// Mitsubishi GX Works2 project: PLC_GROUP_02   PLC: FX3G
// PLC_GROUP_02

// global labels: Global1
VAR_GLOBAL
  sw5 AT X005 : BOOL;
  light7 AT Y007 : BOOL;
  ts1 AT TS1 : BOOL;
  light1 AT Y001 : BOOL;
  ts2 AT TS2 : BOOL;
  inventoryRaspberry AT D1102 : INT;
  inventoryLemon AT D1104 : INT;
  inventoryStabilizer AT D1106 : INT;
  inventoryGummy AT D1108 : INT;
  sw3 AT X003 : BOOL;
  light2 AT Y002 : BOOL;
  anlogInput1 AT D8280 : INT;
  helper11 AT M11 : ARRAY [0..2] OF BOOL;
  regularGummy AT M12 : BOOL;
  luxeryGummy AT M13 : BOOL;
  tc1 AT TC1 : BOOL;
  tempDetected AT M5 : BOOL;
  tc2 AT TC2 : BOOL;
END_VAR
VAR_GLOBAL CONSTANT
  constant0 : INT;
  constant5 : INT := 5;
END_VAR
VAR_GLOBAL
  light0 AT Y000 : BOOL;
END_VAR
VAR_GLOBAL CONSTANT
  needRaspberryReg : INT := 280;
  needLemonReg : INT := 455;
  needStabilizerReg : INT := 105;
  needGummyReg : INT := 28;
  needRaspberryLux : INT := 385;
  needLemonLux : INT := 665;
  needStabilizerLux : INT := 210;
  needGummyLux : INT := 70;
  lemonAndRaspberryMake : INT := 10;
  LemRasMaking : INT := 50;
END_VAR
VAR_GLOBAL
  cooling AT X002 : BOOL;
  temp AT D1130 : INT;
END_VAR
VAR_GLOBAL CONSTANT
  twoCoolingTime : INT := 160;
  onePackage : INT := 1;
  byTen : REAL := 10.0;
END_VAR
VAR_GLOBAL
  inventory AT M1 : BOOL;
  emergency AT X005 : BOOL;
  chooseType AT X001 : BOOL;
  determineType AT M11 : ARRAY [0..2] OF BOOL;
  noInvantoryRegular AT M4 : BOOL;
  noInvantoryLux AT M6 : BOOL;
  tempSensor AT X003 : BOOL;
  startD AT X007 : BOOL;
  helper0 AT M0 : BOOL;
  ts3 AT TS3 : BOOL;
  tc3 AT TC3 : BOOL;
END_VAR
VAR_GLOBAL CONSTANT
  mixingTimeReg : INT := 30;
END_VAR
VAR_GLOBAL
  light5 AT Y005 : BOOL;
  ts4 AT TS4 : BOOL;
  light6 AT Y006 : BOOL;
  tc4 AT TC4 : BOOL;
  tc5 AT TC5 : BOOL;
  tc6 AT TC6 : BOOL;
END_VAR
VAR_GLOBAL CONSTANT
  mixingTimelux : INT := 50;
END_VAR
VAR_GLOBAL
  ts5 AT TS5 : BOOL;
  ts6 AT TS6 : BOOL;
END_VAR
VAR_GLOBAL CONSTANT
  flickeringTime : INT := 5;
END_VAR
VAR_GLOBAL
  last AT M13 : BOOL;
  first AT M1 : BOOL;
  restAllM AT M14 : BOOL;
END_VAR
VAR_GLOBAL CONSTANT
  lessThen5 : INT := 5;
  con0 : INT;
  con5 : INT := 5;
  con6 : INT := 6;
  con10 : INT := 10;
  conFlote10 : REAL := 10.0;
  con40 : INT := 40;
  con400 : INT := 400;
END_VAR
VAR_GLOBAL
  sampleInput AT M2 : BOOL;
  endOfDay AT M3 : BOOL;
  analogOut AT D8282 : INT;
  packages AT D1130 : INT;
  endOfDaytPack AT D1132 : INT;
  analogInputDiv AT D1140 : INT;
  coolingCont AT D1142 : INT;
END_VAR
VAR_GLOBAL CONSTANT
  rasRegGram : INT := 350;
END_VAR
VAR_GLOBAL
  finishFirstCooling AT M7 : BOOL;
END_VAR
VAR_GLOBAL CONSTANT
  limRegGram : INT := 490;
  coolingTime : INT := 80;
END_VAR
VAR_GLOBAL
  mixingCont AT D1144 : INT;
END_VAR
VAR_GLOBAL CONSTANT
  con868 : INT := 868;
  con1330 : INT := 1330;
END_VAR
VAR_GLOBAL
  coolingContRas AT D1142 : INT;
  coolingContlim AT D1146 : INT;
END_VAR
VAR_GLOBAL CONSTANT
  limLuxGram : INT := 700;
  rasLuxGram : INT := 560;
END_VAR
VAR_GLOBAL
  stopDay AT M20 : BOOL;
  firstD AT D1102 : INT;
  lastD AT D1130 : INT;
  first2D AT D1134 : INT;
  last2D AT D1146 : INT;
  startMixing AT M8 : BOOL;
END_VAR

// task Task_01 (event TRUE, interval 0, priority 31): POU_01

PROGRAM POU_01
(* structured ladder/FBD written out as ST: instructions are called as NAME(EN, inputs, outputs); _pN, _eN, _tN stand for wires *)
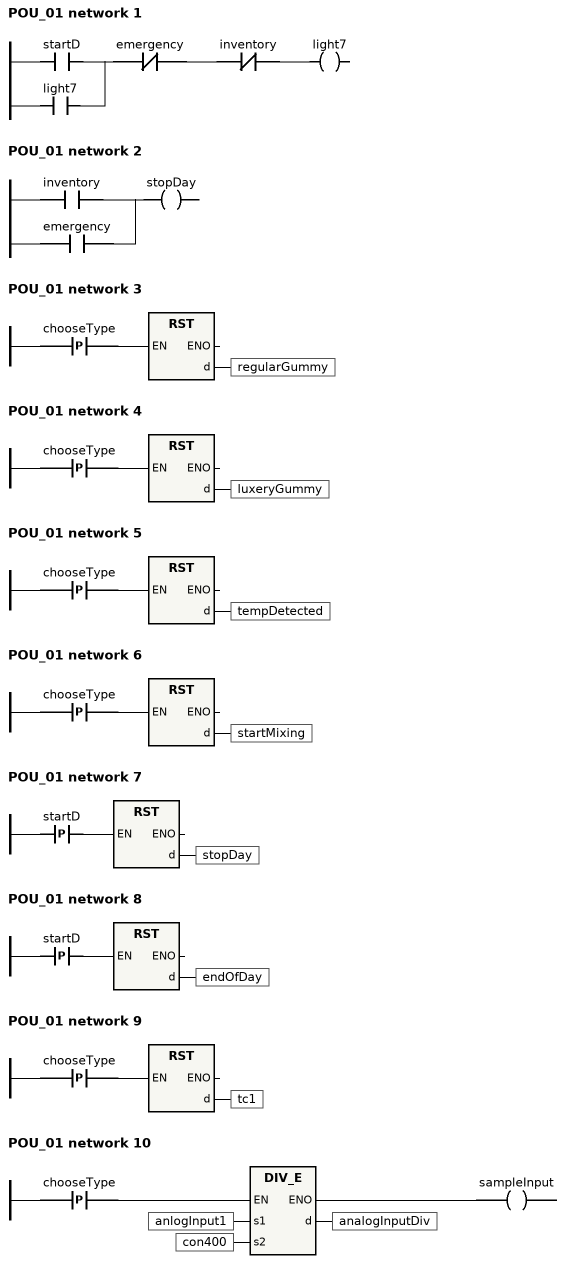
(* network 1 *)
light7 := ((startD OR light7) AND NOT emergency) AND NOT inventory;
(* network 2 *)
stopDay := inventory OR emergency;
(* network 3 *)
RST(LDP(TRUE, chooseType), regularGummy);
(* network 4 *)
RST(LDP(TRUE, chooseType), luxeryGummy);
(* network 5 *)
RST(LDP(TRUE, chooseType), tempDetected);
(* network 6 *)
RST(LDP(TRUE, chooseType), startMixing);
(* network 7 *)
RST(LDP(TRUE, startD), stopDay);
(* network 8 *)
RST(LDP(TRUE, startD), endOfDay);
(* network 9 *)
RST(LDP(TRUE, chooseType), tc1);
(* network 10 *)
_e1 := DIV_E(LDP(TRUE, chooseType), anlogInput1, con400, analogInputDiv);
sampleInput := _e1;
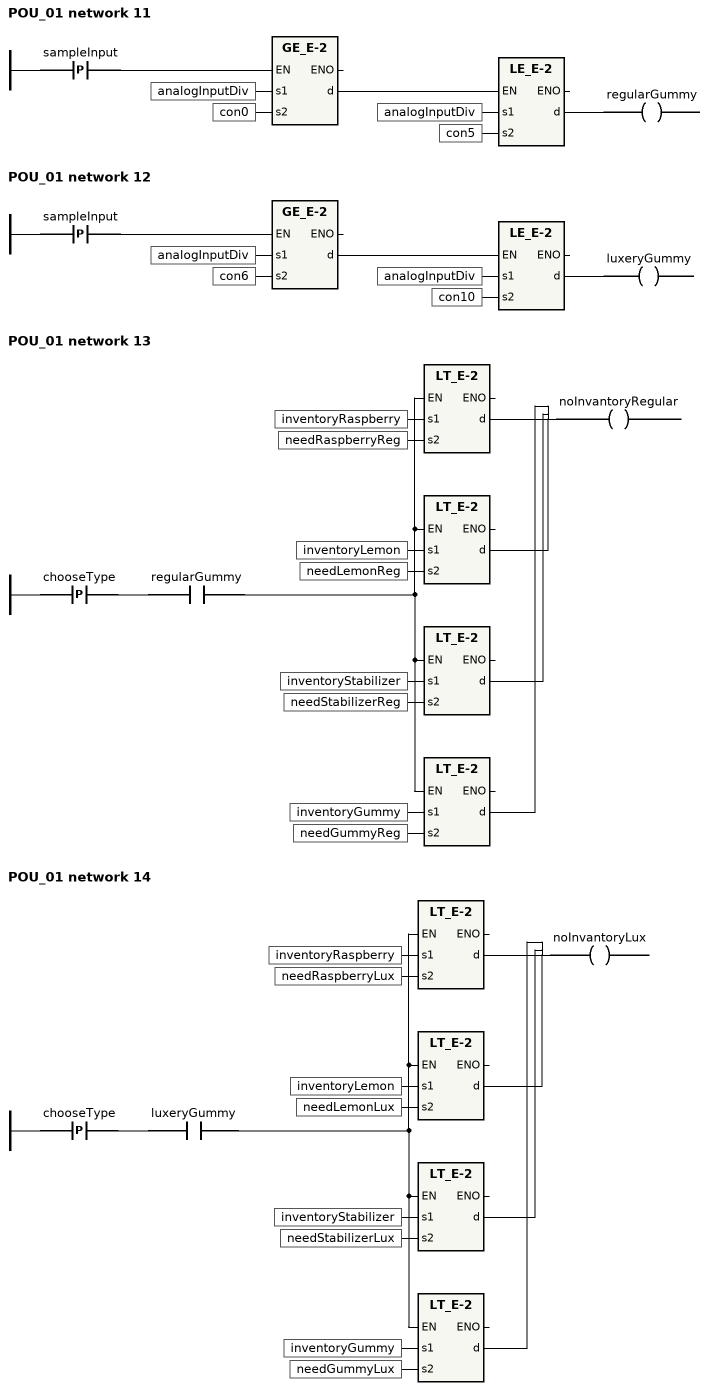
(* network 11 *)
GE_E(LDP(TRUE, sampleInput), analogInputDiv, con0, _t1);
LE_E(_t1, analogInputDiv, con5, _t2);
regularGummy := _t2;
(* network 12 *)
GE_E(LDP(TRUE, sampleInput), analogInputDiv, con6, _t1);
LE_E(_t1, analogInputDiv, con10, _t2);
luxeryGummy := _t2;
(* network 13 *)
_p1 := LDP(TRUE, chooseType) AND regularGummy;
LT_E(_p1, inventoryRaspberry, needRaspberryReg, _t2);
LT_E(_p1, inventoryLemon, needLemonReg, _t3);
LT_E(_p1, inventoryStabilizer, needStabilizerReg, _t4);
LT_E(_p1, inventoryGummy, needGummyReg, _t5);
noInvantoryRegular := _t2 OR _t3 OR _t4 OR _t5;
(* network 14 *)
_p1 := LDP(TRUE, chooseType) AND luxeryGummy;
LT_E(_p1, inventoryRaspberry, needRaspberryLux, _t2);
LT_E(_p1, inventoryLemon, needLemonLux, _t3);
LT_E(_p1, inventoryStabilizer, needStabilizerLux, _t4);
LT_E(_p1, inventoryGummy, needGummyLux, _t5);
noInvantoryLux := _t2 OR _t3 OR _t4 OR _t5;
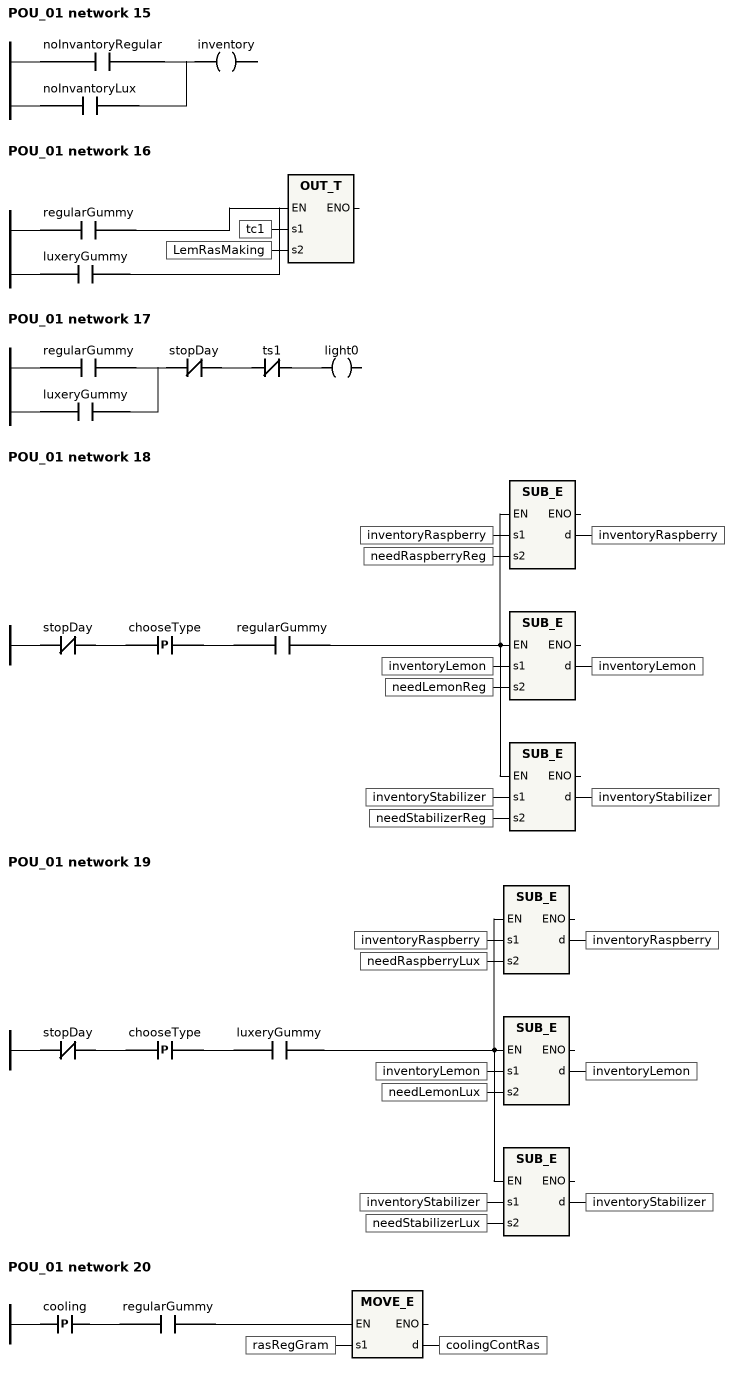
(* network 15 *)
inventory := noInvantoryRegular OR noInvantoryLux;
(* network 16 *)
OUT_T(regularGummy OR luxeryGummy, tc1, LemRasMaking);
(* network 17 *)
light0 := ((regularGummy OR luxeryGummy) AND NOT stopDay) AND NOT ts1;
(* network 18 *)
_p1 := NOT stopDay AND LDP(TRUE, chooseType) AND regularGummy;
SUB_E(_p1, inventoryRaspberry, needRaspberryReg, inventoryRaspberry);
SUB_E(_p1, inventoryLemon, needLemonReg, inventoryLemon);
SUB_E(_p1, inventoryStabilizer, needStabilizerReg, inventoryStabilizer);
(* network 19 *)
_p1 := NOT stopDay AND LDP(TRUE, chooseType) AND luxeryGummy;
SUB_E(_p1, inventoryRaspberry, needRaspberryLux, inventoryRaspberry);
SUB_E(_p1, inventoryLemon, needLemonLux, inventoryLemon);
SUB_E(_p1, inventoryStabilizer, needStabilizerLux, inventoryStabilizer);
(* network 20 *)
MOVE_E(LDP(TRUE, cooling) AND regularGummy, rasRegGram, coolingContRas);
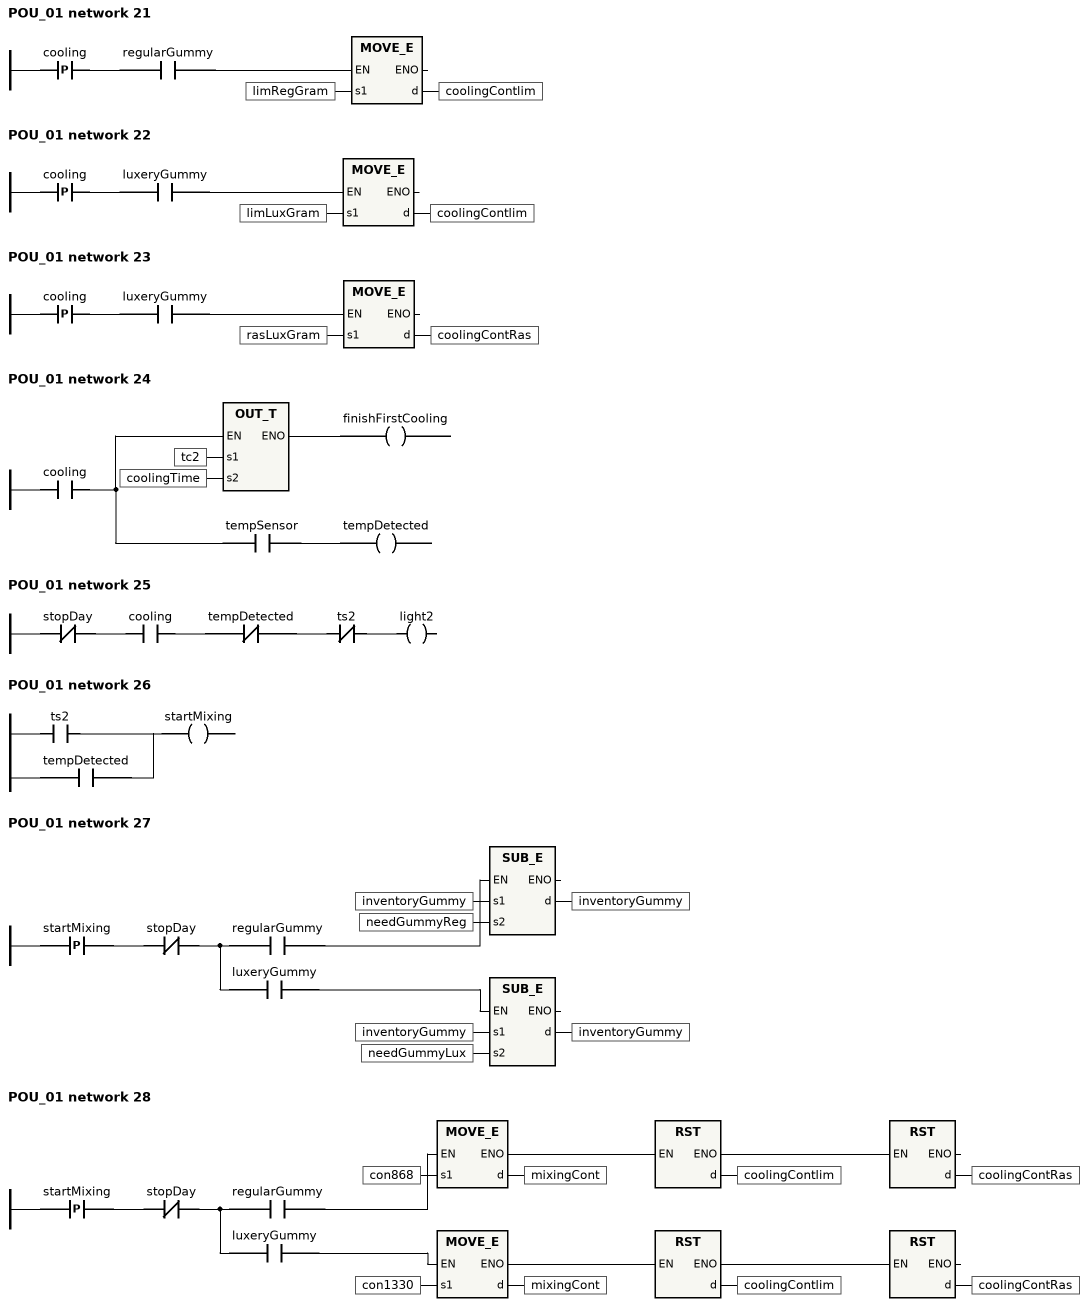
(* network 21 *)
MOVE_E(LDP(TRUE, cooling) AND regularGummy, limRegGram, coolingContlim);
(* network 22 *)
MOVE_E(LDP(TRUE, cooling) AND luxeryGummy, limLuxGram, coolingContlim);
(* network 23 *)
MOVE_E(LDP(TRUE, cooling) AND luxeryGummy, rasLuxGram, coolingContRas);
(* network 24 *)
_e1 := OUT_T(cooling, tc2, coolingTime);
finishFirstCooling := _e1;
tempDetected := cooling AND tempSensor;
(* network 25 *)
light2 := NOT stopDay AND cooling AND NOT tempDetected AND NOT ts2;
(* network 26 *)
startMixing := ts2 OR tempDetected;
(* network 27 *)
_p1 := LDP(TRUE, startMixing) AND NOT stopDay;
SUB_E(_p1 AND regularGummy, inventoryGummy, needGummyReg, inventoryGummy);
SUB_E(_p1 AND luxeryGummy, inventoryGummy, needGummyLux, inventoryGummy);
(* network 28 *)
_p1 := LDP(TRUE, startMixing) AND NOT stopDay;
_e2 := MOVE_E(_p1 AND regularGummy, con868, mixingCont);
_e3 := RST(_e2, coolingContlim);
RST(_e3, coolingContRas);
_e4 := MOVE_E(_p1 AND luxeryGummy, con1330, mixingCont);
_e5 := RST(_e4, coolingContlim);
RST(_e5, coolingContRas);
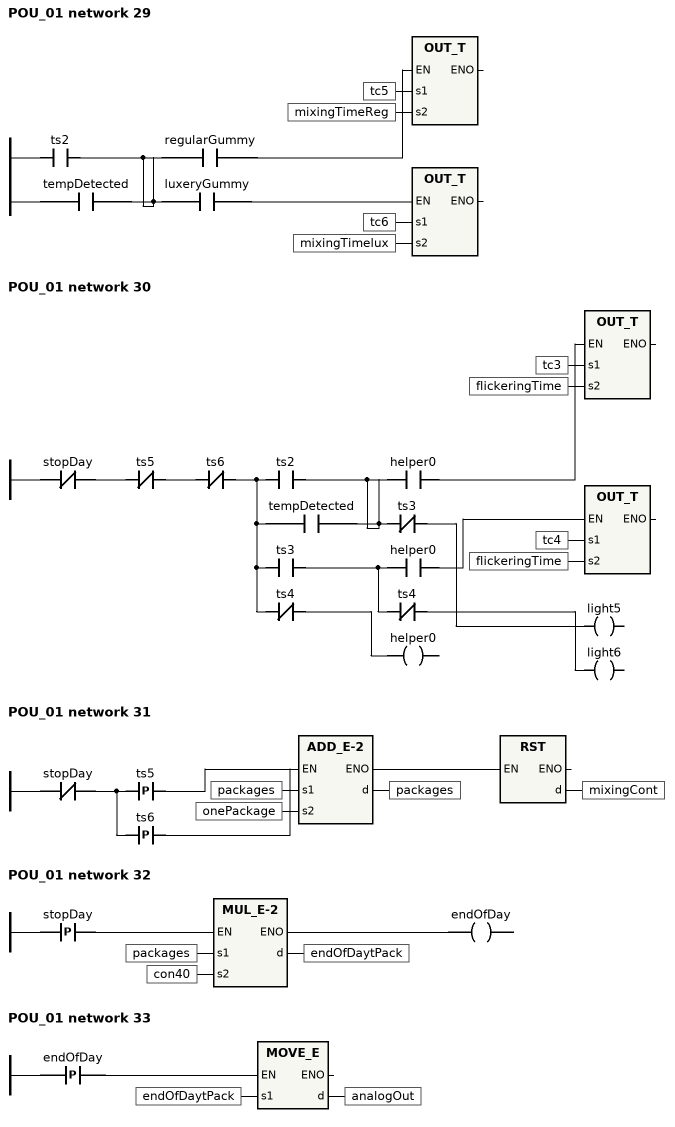
(* network 29 *)
_p1 := ts2 OR tempDetected;
OUT_T(_p1 AND regularGummy, tc5, mixingTimeReg);
OUT_T(_p1 AND luxeryGummy, tc6, mixingTimelux);
(* network 30 *)
_p1 := NOT stopDay AND NOT ts5 AND NOT ts6;
_p2 := (_p1 AND ts2) OR (_p1 AND tempDetected);
OUT_T(_p2 AND helper0, tc3, flickeringTime);
light5 := _p2 AND NOT ts3;
_p3 := _p1 AND ts3;
OUT_T(_p3 AND helper0, tc4, flickeringTime);
light6 := _p3 AND NOT ts4;
helper0 := _p1 AND NOT ts4;
(* network 31 *)
_p1 := NOT stopDay;
_e2 := ADD_E((_p1 AND LDP(TRUE, ts5)) OR (_p1 AND LDP(TRUE, ts6)), packages, onePackage, packages);
RST(_e2, mixingCont);
(* network 32 *)
_e1 := MUL_E(LDP(TRUE, stopDay), packages, con40, endOfDaytPack);
endOfDay := _e1;
(* network 33 *)
MOVE_E(LDP(TRUE, endOfDay), endOfDaytPack, analogOut);
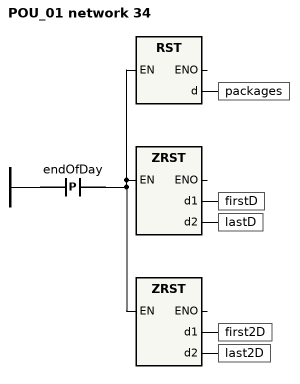
(* network 34 *)
_p1 := LDP(TRUE, endOfDay);
RST(_p1, packages);
ZRST(_p1, firstD, lastD);
ZRST(_p1, first2D, last2D);
END_PROGRAM
